Fanuc KAREL source: kb00067.KL

-- PROVISIONAL review KL for V940-1; original PC SHA256 9285984c054e630718d4c8685cb326e45417c339dfd75118d1cd97a7b4181ef8
-- Incomplete behavior may be omitted. Consult companion uncertainty JSON. Do not deploy.
PROGRAM KB00067
%NOLOCKGROUP
BEGIN
  -- V9_ZERO_TABLE_METADATA_HINT layout=0002_ascii; no indexed target words; source/name/runtime held
  -- UNRESOLVED_PC offsets 5-14; opcodes 3F,75
  -- UNRESOLVED_PC offsets 19-26; opcodes 9D,23
  -- UNRESOLVED_PC offsets 31-38; opcodes 9D,23
  -- UNRESOLVED_PC offsets 43-50; opcodes 9D,23
  -- UNRESOLVED_PC offsets 55-62; opcodes 9D,23
  -- UNRESOLVED_PC offsets 67-103; opcodes 27,22,2A,22,22,22,22,31
  -- UNRESOLVED_PC offsets 108-112; opcodes 7F
END KB00067
